FUNCTION_BLOCK EL1014
VAR
	_io : EL1xx4_Data;
	{attribute addProperty Name "WcState"}
	_wcState : WcStateInputToggle;
	{attribute addProperty Name "Info data"}
	_infoData : InfoDataBase;
END_VAR

PROPERTY IO : REFERENCE TO EL1xx4_Data
GET
IO REF= _io;
END_GET
END_PROPERTY

PROPERTY WcState : REFERENCE TO WcStateInputToggle
GET
WcState REF= _wcState;
END_GET
END_PROPERTY

END_FUNCTION_BLOCK

(* stored: Version 1.1.0.1, ProductVersion 3.1.4024.9
   POU EL1014: Id {691bb5d3-23e2-0ad4-2d95-81127c263eda}, SpecialFunc None
   Property IO: Id {ddbf1984-07e5-0eba-0c19-236dceff503e}
   Get Get: Id {06626c43-1791-046b-15a9-724cfa5dd8a2}
   Property WcState: Id {57d493f1-2522-0c75-1edd-5999fab3520b}
   Get Get: Id {c0422d43-a05c-0804-1b42-a18c2cf1e8db} *)
